TYPE ST_VisControl :
STRUCT
	
	stControlPad	: ST_Vis_ControlPadControl;
	stOperatorPad	: ST_Vis_OperationalControl;


END_STRUCT
END_TYPE

(* stored: Version 1.1.0.1, ProductVersion 3.1.4024.4
   DUT ST_VisControl: Id {c330307e-d464-4336-b6c6-600891ee7229} *)
